// TIA Portal project "spsNeu" (V16)

(* hardware
DEVICE "S7-1200-Station_1"  S7-1200 Station
   slot 0: "Baugruppenträger_0"  S7-1200 Rack  Rack  V1.0
   slot 1: "PLC_1"  CPU 1214C DC/DC/DC  6ES7 214-1AG40-0XB0  V4.4
*)

// ===== PLC "PLC_1"  CPU 1214C DC/DC/DC =====

VAR_GLOBAL   // PLC tag table "Standard-Variablentabelle"
   "Motor_links" AT %Q0.0 : Bool;
   "Motor_rechts" AT %Q0.1 : Bool;
   "OUT3" AT %Q0.2 : Bool;
   "IN1" AT %I0.0 : Bool;
   "IN2" AT %I0.1 : Bool;
   "IN3" AT %I0.2 : Bool;
   "Sim_ID1000" AT %I1.0 : Bool;
END_VAR

DATA_BLOCK "Datenbaustein_1"   // DB1
{ S7_Optimized_Access := 'FALSE' }
VERSION : 0.1
   VAR
      Webserver : Struct
         Job_ID : Int;
         Start_Job : Bool;
      END_STRUCT;
      Foerderband : Struct
         Sensor : Struct
            B1 : Bool;   // Sensor Einlauf Förderband [NO]
            B2 : Bool;   // Sensor Auslauf Förderband [NO]
         END_STRUCT;
         Motor : Struct
            links : Bool;
            rechts : Bool;
         END_STRUCT;
      END_STRUCT;
      HMI : Struct
         Bedienfeld : Struct
            Taster : Struct
               EIN : Bool;
            END_STRUCT;
         END_STRUCT;
      END_STRUCT;
   END_VAR
BEGIN
END_DATA_BLOCK

ORGANIZATION_BLOCK "Main"   // OB1, FBD, ProgramCycle
TITLE = "Main Program Sweep (Cycle)"
{ S7_Optimized_Access := 'TRUE' }
VERSION : 0.1
   VAR_INPUT
      Initial_Call : Bool;   // Initial call of this OB
      Remanence : Bool;   // =True, if remanent data are available
   END_VAR
BEGIN

REGION Network 1
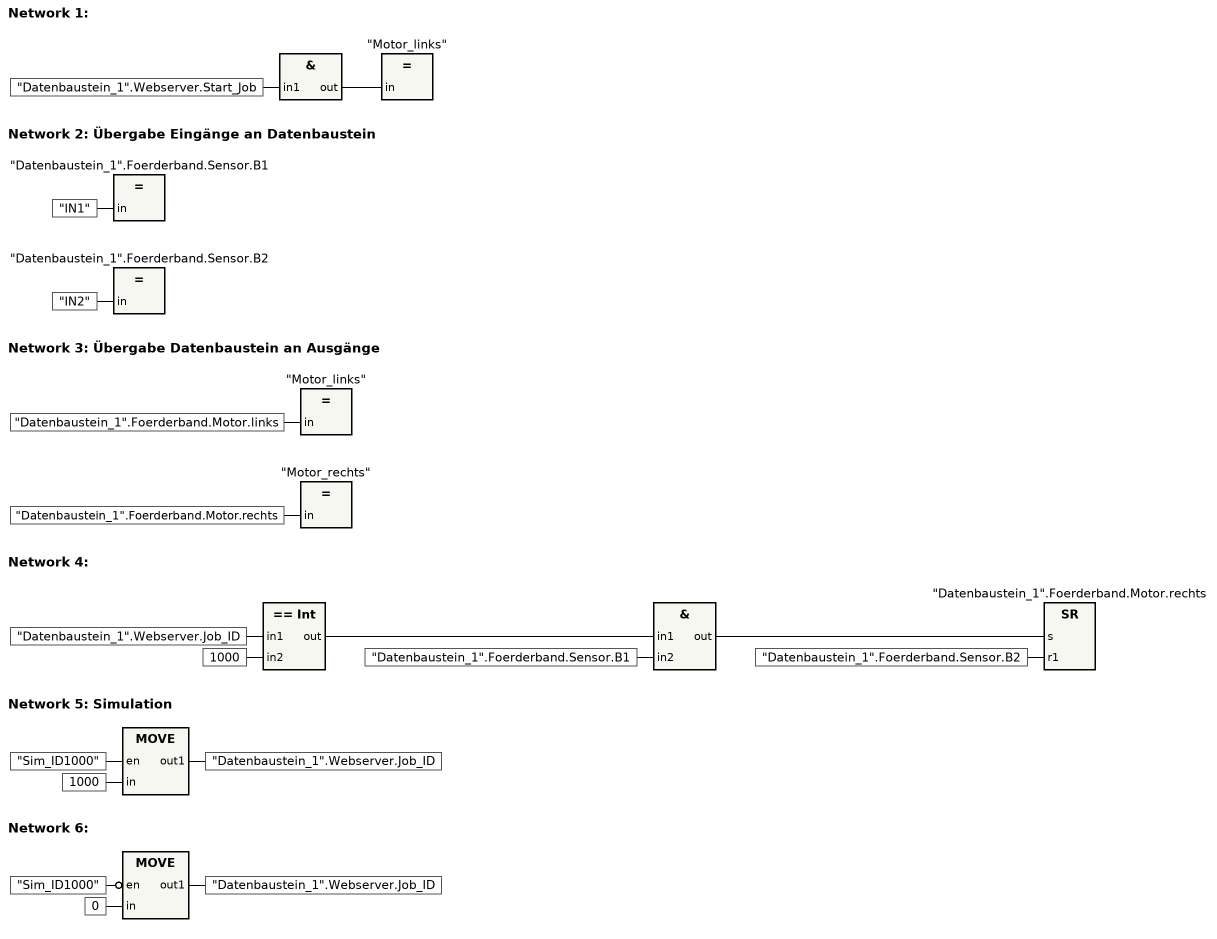
   "Motor_links" := "Datenbaustein_1".Webserver.Start_Job;
END_REGION

REGION Network 2: Übergabe Eingänge an Datenbaustein
   "Datenbaustein_1".Foerderband.Sensor.B1 := "IN1";
   "Datenbaustein_1".Foerderband.Sensor.B2 := "IN2";
END_REGION

REGION Network 3: Übergabe Datenbaustein an Ausgänge
   "Motor_links" := "Datenbaustein_1".Foerderband.Motor.links;
   "Motor_rechts" := "Datenbaustein_1".Foerderband.Motor.rechts;
END_REGION

REGION Network 4
   IF ("Datenbaustein_1".Webserver.Job_ID = 1000) AND "Datenbaustein_1".Foerderband.Sensor.B1 THEN
       "Datenbaustein_1".Foerderband.Motor.rechts := TRUE;   // SR flip-flop
   END_IF;
   IF "Datenbaustein_1".Foerderband.Sensor.B2 THEN
       "Datenbaustein_1".Foerderband.Motor.rechts := FALSE;
   END_IF;
END_REGION

REGION Network 5: Simulation
   IF "Sim_ID1000" THEN "Datenbaustein_1".Webserver.Job_ID := 1000; END_IF;
END_REGION

REGION Network 6
   IF NOT "Sim_ID1000" THEN "Datenbaustein_1".Webserver.Job_ID := 0; END_IF;
END_REGION
END_ORGANIZATION_BLOCK